Yaskawa INFORM job: pos_x_0.JBI

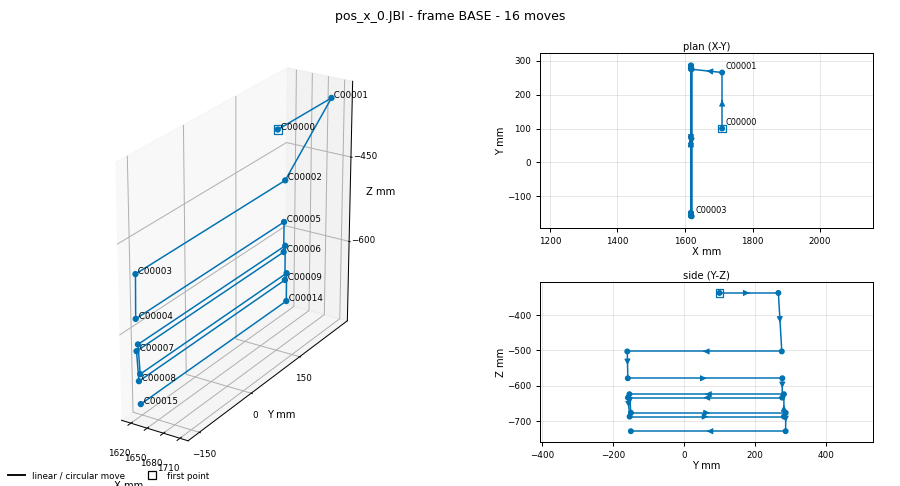
[picture p0: tool path of pos_x_0.JBI in frame BASE, 16 of 18 moves have a stored position in this frame; points joined in program order, loops and branches not executed]
/JOB
//NAME pos_x_0
//POS
///NPOS 16,0,16,0,0,0
///TOOL 0
///POSTYPE BASE
///RECTAN
///RCONF 0,0,0,0,0,0,0,0,0,0,0,0,0,0,0,0,0,0,0,0,0,0,0,0
C00000=1709.879320,99.983217,-337.785080,180.000000,-89.999999,0.000000
C00001=1709.879320,265.846217,-337.785080,180.000000,-89.999999,0.000000
C00002=1619.762523,275.472038,-502.616041,180.000000,-89.999999,0.000000
C00003=1619.762523,-160.131962,-502.616041,180.000000,-89.999999,0.000000
C00004=1617.419464,-158.625922,-578.294103,180.000000,-89.999999,0.000000
C00005=1617.419464,276.980078,-578.294103,180.000000,-89.999999,0.000000
C00006=1617.352670,276.615658,-632.957507,180.000000,-89.999999,0.000000
C00007=1617.352670,-158.159342,-632.957507,180.000000,-89.999999,0.000000
C00008=1617.369708,-153.446402,-686.390485,180.000000,-89.999999,0.000000
C00009=1617.369708,281.436598,-686.390485,180.000000,-89.999999,0.000000
C00010=1617.417708,281.411239,-623.243274,180.000000,-60.000000,0.000000
C00011=1617.417708,-154.047761,-623.243274,180.000000,-60.000000,0.000000
C00012=1617.499943,-149.907339,-675.747370,180.000000,-60.000000,0.000000
C00013=1617.499943,286.549561,-675.747370,180.000000,-60.000000,0.000000
C00014=1617.585020,286.293971,-727.548848,180.000000,-60.000000,0.000000
C00015=1617.585020,-150.003529,-727.548848,180.000000,-60.000000,0.000000
///POSTYPE PULSE
///PULSE
EX000=276480
///POSTYPE PULSE
///PULSE
EC00000=276480
EC00001=276480
EC00002=276480
EC00003=276480
EC00004=276480
EC00005=276480
EC00006=276480
EC00007=276480
EC00008=276480
EC00009=276480
EC00010=276480
EC00011=276480
EC00012=276480
EC00013=276480
EC00014=276480
EC00015=276480
//INST
///DATE 2023/06/26 11:09
///ATTR SC,RW,RJ
////FRAME BASE
///GROUP1 RB1,ST1
NOP
MOVJ P009 EX000 VJ=15.00
MOVJ C00000 EC00000 VJ=15.0
CALL JOB:SPYON
MOVL C00001 EC00001 V=150.0
MOVL C00002 EC00002 V=150.0
MOVL C00003 EC00003 V=150.0
MOVL C00004 EC00004 V=150.0
MOVL C00005 EC00005 V=150.0
MOVL C00006 EC00006 V=150.0
MOVL C00007 EC00007 V=150.0
MOVL C00008 EC00008 V=150.0
MOVL C00009 EC00009 V=150.0
MOVL C00010 EC00010 V=150.0
MOVL C00011 EC00011 V=150.0
MOVL C00012 EC00012 V=150.0
MOVL C00013 EC00013 V=150.0
MOVL C00014 EC00014 V=150.0
MOVL C00015 EC00015 V=150.0
CALL JOB:SPYOF
MOVJ P009 VJ=15.00
END
